PROGRAM AxisController
VAR
	directionVertical : BOOL;
	positionVertical : INT;
	EncoderSignalProcessor_Vertical: EncoderSignalProcessor;
	initialPosition: INT := 0;
	EncoderSignalProcessor_Horizontal: EncoderSignalProcessor;
	positionHorizontal: INT;
	directionHorizontal: BOOL;
	positionRotational: INT;
	directionRotational: BOOL;
	EncoderSignalProcessor_Rotational: EncoderSignalProcessor;
END_VAR

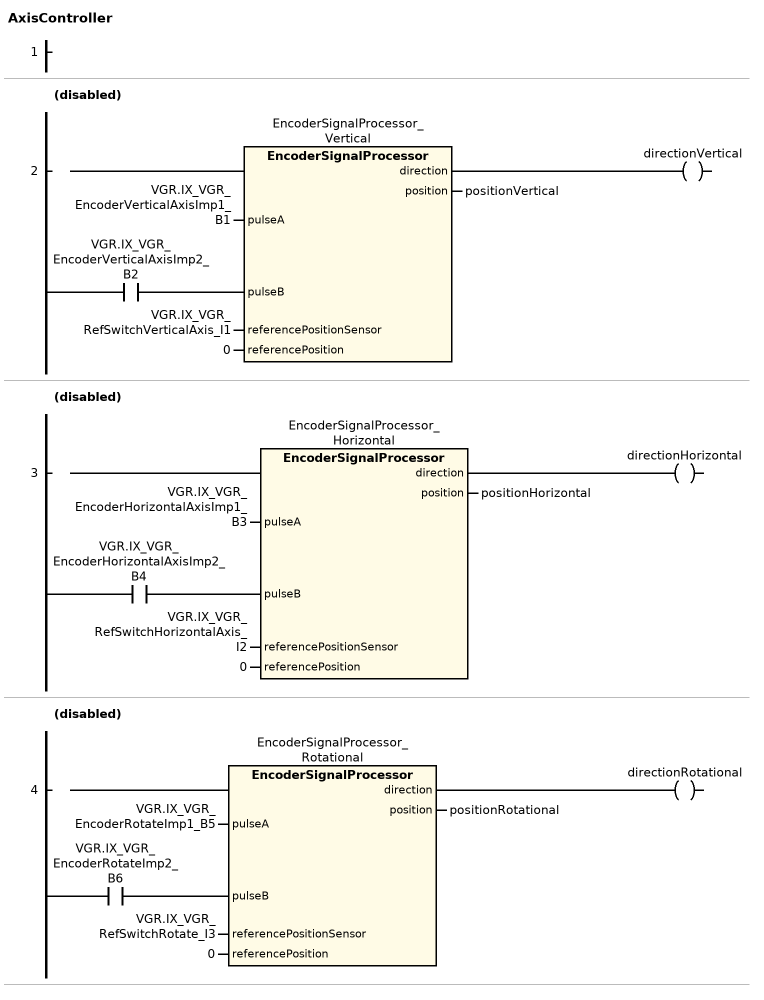
// NETWORK 1

// NETWORK 2 (disabled)
// EncoderSignalProcessor_Vertical(
//     pulseA := VGR.IX_VGR_EncoderVerticalAxisImp1_B1,
//     pulseB := VGR.IX_VGR_EncoderVerticalAxisImp2_B2,
//     referencePositionSensor := VGR.IX_VGR_RefSwitchVerticalAxis_I1,
//     referencePosition := 0,
//     position => positionVertical); // EncoderSignalProcessor
// directionVertical := EncoderSignalProcessor_Vertical.direction;

// NETWORK 3 (disabled)
// EncoderSignalProcessor_Horizontal(
//     pulseA := VGR.IX_VGR_EncoderHorizontalAxisImp1_B3,
//     pulseB := VGR.IX_VGR_EncoderHorizontalAxisImp2_B4,
//     referencePositionSensor := VGR.IX_VGR_RefSwitchHorizontalAxis_I2,
//     referencePosition := 0,
//     position => positionHorizontal); // EncoderSignalProcessor
// directionHorizontal := EncoderSignalProcessor_Horizontal.direction;

// NETWORK 4 (disabled)
// EncoderSignalProcessor_Rotational(
//     pulseA := VGR.IX_VGR_EncoderRotateImp1_B5,
//     pulseB := VGR.IX_VGR_EncoderRotateImp2_B6,
//     referencePositionSensor := VGR.IX_VGR_RefSwitchRotate_I3,
//     referencePosition := 0,
//     position => positionRotational); // EncoderSignalProcessor
// directionRotational := EncoderSignalProcessor_Rotational.direction;

END_PROGRAM

(* stored: Version 1.1.0.1, ProductVersion 3.1.4024.12
   POU AxisController: Id {11839d6a-824f-4210-8327-a23f96ebc9d2}, SpecialFunc None *)
